(* IEC 61131-3 sources: Std_PalletMover/Class/MqttTopicText, 1 file *)

(* ---- MqttTopicText.st ---- *)
(*!
<Class
	Name               = "MqttTopicText"
	Revision           = "0.0"
	RealtimeTask       = "false"
	CyclicTask         = "true"
	BackgroundTask     = "false"
	Sigmatek           = "false"
	OSInterface        = "false"
	HighPriority       = "false"
	Automatic          = "false"
	UpdateMode         = "Prescan"
	SharedCommandTable = "true"
	Objectsize         = "(730,120)">
	<Channels>
		<Server Name="DataReceived" Visualized="false" Initialize="false" WriteProtected="true" Retentive="false"/>
		<Server Name="EnableMessage" Visualized="false" Initialize="true" WriteProtected="false" Retentive="File"/>
		<Client Name="objRiwoEventLogger" Required="false" Internal="false"/>
	</Channels>
	<Network Name="MqttTopicText">
		<!-- List of Components in this network -->
		<Components>
			<Object
				Name       = "_base"
				Class      = "MQTTTopicString"
				Position   = "(218,120)"
				Visualized = "true"
				Remotely   = "true">
				<Channels>
					<Server Name="DataString"/>
					<Server Name="GrantedQoS"/>
					<Server Name="PublishInterval" Value="10 sec"/>
					<Server Name="QoS"/>
					<Server Name="RetainData"/>
					<Server Name="TopicName"/>
					<Server Name="TopicState"/>
					<Server Name="TopicType"/>
					<Client Name="cAutoResetTime" Value="MQTTTOPIC_DEFAULT_AUTORESET_TIME"/>
					<Client Name="cPublishTimeout" Value="MQTTTOPIC_DEFAULT_PUBLISH_TIMEOUT"/>
					<Client Name="cSubscribeTimeout" Value="MQTTTOPIC_DEFAULT_SUBSCRIBE_TIMEOUT"/>
					<Client Name="cUnsubscribeTimeout" Value="MQTTTOPIC_DEFAULT_UNSUBSCRIBE_TIMEOUT"/>
					<Client Name="ocMQTTClient_Interface"/>
					<Client Name="ocSigCLib"/>
					<Client Name="ocStdLib"/>
				</Channels>
			</Object>
		</Components>
		<Comments>
		</Comments>
		<!-- List of Connections in this network -->
		<Connections>
			<Connection Source="this.TopicState" Destination="_base.TopicState" Vertices="(2236,210),(2064,210),"/>
			<Connection Source="this.TopicType" Destination="_base.TopicType" Vertices="(2236,270),(2064,270),"/>
			<Connection Source="this.TopicName" Destination="_base.TopicName" Vertices="(2236,330),(2064,330),"/>
			<Connection Source="this.PublishInterval" Destination="_base.PublishInterval" Vertices="(2236,390),(2064,390),"/>
			<Connection Source="this.RetainData" Destination="_base.RetainData" Vertices="(2236,450),(2064,450),"/>
			<Connection Source="this.QoS" Destination="_base.QoS" Vertices="(2236,510),(2064,510),"/>
			<Connection Source="this.GrantedQoS" Destination="_base.GrantedQoS" Vertices="(2236,570),(2064,570),"/>
			<Connection Source="this.DataString" Destination="_base.DataString" Vertices="(2236,630),(2064,630),"/>
			<Connection Source="_base.ocMQTTClient_Interface" Destination="this.ocMQTTClient_Interface" Vertices="(218,210),(38,210),"/>
		</Connections>
		<!-- Headerfiles -->
		<Options>
		</Options>
	</Network>
</Class>
*)
#pragma using MQTTTopicString

MqttTopicText : CLASS
: MQTTTopicString
  //Servers:
	DataReceived 	: SvrCh_DINT;
	EnableMessage 	: SvrCh_DINT;
  //Clients:
	objRiwoEventLogger 	: CltChCmd_RiwoEventLogger;
  //Variables:
  //Functions:
				//! <Function Comment="Will be called if data from the subscribed topic was received.&#13;&#10;&#13;&#10;Note: the pointer to the data is only valid in the actual call of this method." Name="User_SubscribeData"/>
	FUNCTION VIRTUAL User_SubscribeData
		VAR_INPUT
			pData 	: ^void;			//! <Variable Comment="Pointer to the payload of the MQTT message, if data is available. Otherwise the pointer is NIL." Name="User_SubscribeData.pData"/>
			udLen 	: UDINT;			//! <Variable Comment="Size of the data in byte." Name="User_SubscribeData.udLen"/>
		END_VAR;

	FUNCTION GLOBAL SetText
		VAR_INPUT
			pText 	: ^CHAR;
		END_VAR;

	FUNCTION GLOBAL GetPublishedFlag
		VAR_OUTPUT
			returnValue 	: BOOL;
		END_VAR;

	FUNCTION GLOBAL GetTopicState
		VAR_OUTPUT
			returnValue 	: t_e_MQTT_TopicState;
		END_VAR;

	FUNCTION GLOBAL Reconnect
		VAR_INPUT
			ConnectRequest 	: DINT;
		END_VAR;

	FUNCTION GLOBAL SetTopicName
		VAR_INPUT
			input 	: ^CHAR;
		END_VAR;

	FUNCTION GLOBAL GetDataString
		VAR_INPUT
			pData 	: ^CHAR;
			dataLength 	: UDINT;
		END_VAR
		VAR_OUTPUT
			returnValue 	: UDINT;
		END_VAR;
  //Tables:
	FUNCTION @STD
		VAR_OUTPUT
			ret_code	: CONFSTATES;
		END_VAR;
	FUNCTION GLOBAL TAB @CT_;
END_CLASS;

#pragma usingLtd RiwoEventLogger

FUNCTION GLOBAL MqttTopicText::SetText
	VAR_INPUT
		pText 	: ^CHAR;
	END_VAR

  if pText <> nil then
    PubSubDataString.WriteDataOff(udLen :=  _strlen(src:=pText),
                                  udOff :=  0,
                                  pData :=  pText);
  else
    _RIWO_ERROR_MSG("Received nil pointer in function MqttTopicText");
  end_if;

END_FUNCTION

FUNCTION GLOBAL MqttTopicText::GetPublishedFlag
	VAR_OUTPUT
		returnValue 	: BOOL;
	END_VAR

  returnValue := FlagList.PublishDone;

END_FUNCTION

FUNCTION GLOBAL MqttTopicText::GetTopicState
	VAR_OUTPUT
		returnValue 	: t_e_MQTT_TopicState;
	END_VAR

  returnValue := TopicState;

END_FUNCTION

FUNCTION GLOBAL MqttTopicText::Reconnect
	VAR_INPUT
		ConnectRequest 	: DINT;
	END_VAR

    if ocMQTTClient_Interface.InterfaceState <> MQTTClient_Interface::MCIS_Connected then
      if ocMQTTClient_Interface.ClientActive = 1 then
        ocMQTTClient_Interface.ClientActive.Write(input:=0); //Reset Client connection
      else
        ocMQTTClient_Interface.ClientActive.Write(input:=1); //Set Client connection
      end_if;
    end_if;

END_FUNCTION

FUNCTION GLOBAL MqttTopicText::SetTopicName
	VAR_INPUT
		input 	: ^CHAR;
	END_VAR

  if input <> nil then
    objTopicName.WriteDataOff(udLen :=  _strlen(src:=input),
                                  udOff :=  0,
                                  pData :=  input);
  else
    _RIWO_ERROR_MSG("Received nil pointer in function MqttTopicText");
  end_if;

END_FUNCTION

FUNCTION GLOBAL MqttTopicText::GetDataString
	VAR_INPUT
		pData 	: ^CHAR;
		dataLength 	: UDINT;
	END_VAR
	VAR_OUTPUT
		returnValue 	: UDINT;
	END_VAR

  if pData <> nil then
    returnValue := PubSubDataString.ReadDataOff(udOff:=0, pData:=pData, udMax:=dataLength);
    DataReceived := false;
  else
    _RIWO_ERROR_MSG("Received nil pointer in function MqttTopicText");
  end_if;

END_FUNCTION

FUNCTION VIRTUAL MqttTopicText::User_SubscribeData
	VAR_INPUT
		pData 	: ^void;
		udLen 	: UDINT;
	END_VAR

  MQTTTopicString::User_SubscribeData(pData,udLen);

  if pData <> nil then
    DataReceived := true;
  else
    _RIWO_ERROR_MSG("Received nil pointer in function MqttTopicText");
  end_if;

END_FUNCTION
